FUNCTION_BLOCK FB_Events EXTENDS FB_Handler
VAR_INPUT
END_VAR
VAR_OUTPUT
END_VAR
VAR
	nEvents:		INT;
	aEvents:		ARRAY [0..100] OF ST_Event;
END_VAR

SUPER^();

METHOD PRIVATE M_Find : INT
VAR_INPUT
	stEvent:			ST_Event;		// event to find
END_VAR
VAR
	nIndex: INT;
END_VAR
FOR nIndex:= 0 TO nEvents DO
	IF memcmp(ADR(aEvents[nEvents]), ADR(stEvent), SIZEOF(stEvent)) = 0 THEN
		M_Find:= nIndex;
		RETURN;
	END_IF
END_FOR
END_METHOD

METHOD PUBLIC M_Request
VAR_INPUT
	stEvent:			ST_Event;		// event to be handled. 
END_VAR
SUPER^.M_Request(stEvent);

IF nEvents < 100 THEN
	IF M_Find(stEvent) = 0 THEN
		aEvents[nEvents]:= stEvent;
		nEvents:= nEvents + 1;
	END_IF
END_IF
END_METHOD

END_FUNCTION_BLOCK

(* stored: Version 1.1.0.1, ProductVersion 3.1.4024.12
   POU FB_Events: Id {a7ae2211-d1a6-49e2-82c8-5c610d8a7c9d}, SpecialFunc None
   Method M_Find: Id {bb4df97c-6e38-4cd5-bdfc-6c0b84052df0}
   Method M_Request: Id {fd7a157e-fd8c-45f8-a7bc-2309e3dc7519} *)
